PROGRAM FUN_ConnectVPN

VAR_INPUT
	ParamNetID				: STRING :='' ; // Unit ID of the PC with internet connexion
	IN_CmdStart 			: BOOL;
	IN_DirExe				: STRING;
	IN_OpenVpnFile			: STRING;
END_VAR
VAR_OUTPUT
	OUT_Completed			: BOOL;
END_VAR

VAR
	RS_Start				: RS;
	TRIG_Completed			: R_TRIG;
	TRIG_Start				: R_TRIG;
	start_process			: NT_StartProcess;
	TRIG_Available			: F_TRIG;
	bTest: BOOL;
END_VAR


TRIG_Start(CLK := IN_CmdStart);

start_process
(
	NETID := ParamNetID,
	PATHSTR := '"C:\Program Files\OpenVPN\bin\openvpn-gui.exe"',
	DIRNAME := 'C:\Program Files\OpenVPN\bin',
	COMNDLINE := Concat(str1 := '--command connect ', str2 := concat(STR1 := IN_OpenVpnFile, STR2 := '.ovpn')),
	Start := TRIG_Start.Q
);

END_PROGRAM

(* stored: Version 1.1.0.1, ProductVersion 3.1.4024.6
   POU FUN_ConnectVPN: Id {4ff0f7b4-9118-4bc6-8c61-19c74f5069a3}, SpecialFunc None *)
